FUNCTION_BLOCK ST_SET_PARM (* Sets the parameter to a data input of a FB, Resource or Device instance *)
  (* Standard: 61499-1; Classification: Reconfiguration; Function: Sets Parameter; Type: Structural Service; Description: Copyright (c) 2012 Profactor GmbH This program and the accompanying materials are made available under the terms of the Eclipse Public License 2.0 which is available at https://www.eclipse.org/legal/epl-2.0/ SPDX-License-Identifier: EPL-2.0 *)
  (* Version 1.0, 2012-05-31, Gerhard Ebenhofer, Profactor GmbH *)
  (* Compiler Cpp GNU GCC >3.0 *)
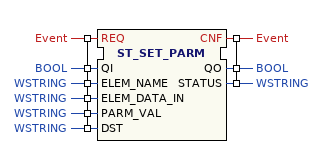
  EVENT_INPUT
    REQ WITH ELEM_NAME, ELEM_DATA_IN, PARM_VAL, DST, QI; (* Event to require setting a parameter *)
  END_EVENT
  EVENT_OUTPUT
    CNF WITH STATUS, QO; (* Event to confirm that the parameter has been set *)
  END_EVENT
  VAR_INPUT
    QI : BOOL; (* Event Input Qualifier *)
    ELEM_NAME : WSTRING; (* Reference to element instance *)
    ELEM_DATA_IN : WSTRING; (* Reference to data input *)
    PARM_VAL : WSTRING; (* Parameter value *)
    DST : WSTRING; (* Destination where the parameter has to be set (Syntax: ResourceName) *)
  END_VAR
  VAR_OUTPUT
    QO : BOOL; (* Event Output Qualifier *)
    STATUS : WSTRING; (* Service Status: RDY, NO_SUCH_OBJECT, INVALID_STATE *)
  END_VAR
END_FUNCTION_BLOCK
